// TIA Portal project "Rid TIA Pick & Place" (V15)
// Vorlageprojekt für das Buch mit Zielsystem S7-1200

(* hardware
DEVICE "S7-1200-Station_1"  S7-1200 Station
   slot 0: "Baugruppenträger_0"  Rack  V1.0
   slot 1: "PLC_1"  CPU 1211C DC/DC/DC  6ES7 211-1AE40-0XB0  V4.1
*)

// ===== PLC "PLC_1"  CPU 1211C DC/DC/DC =====

VAR_GLOBAL   // PLC tag table "Standard-Variablentabelle"
   "Clock_Byte" AT %MB0 : Byte;
   "Clock_10Hz" AT %M0.0 : Bool;
   "Clock_5Hz" AT %M0.1 : Bool;
   "Clock_2.5Hz" AT %M0.2 : Bool;
   "Clock_2Hz" AT %M0.3 : Bool;
   "Clock_1.25Hz" AT %M0.4 : Bool;
   "Clock_1Hz" AT %M0.5 : Bool;
   "Clock_0.625Hz" AT %M0.6 : Bool;
   "Clock_0.5Hz" AT %M0.7 : Bool;
END_VAR

VAR_GLOBAL   // PLC tag table "Assembler"
   "Item at entry" AT %I0.0 : Bool;
   "Item at exit" AT %I0.1 : Bool;
   "Moving X" AT %I0.2 : Bool;
   "Moving Z" AT %I0.3 : Bool;
   "Item detected" AT %I0.4 : Bool;
   "Start" AT %I0.5 : Bool;
   "Reset" AT %I0.6 : Bool;
   "Stop" AT %I0.7 : Bool;
   "Emergency stop" AT %I1.0 : Bool;
   "Auto" AT %I1.1 : Bool;
   "FACTORY I/O (Running)" AT %I1.2 : Bool;
   "Entry conveyor" AT %Q0.0 : Bool;
   "Exit conveyor" AT %Q0.1 : Bool;
   "Move X" AT %Q0.2 : Bool;
   "Move Z" AT %Q0.3 : Bool;
   "Grab" AT %Q0.4 : Bool;
   "Start light" AT %Q0.5 : Bool;
   "Reset light" AT %Q0.6 : Bool;
   "Stop light" AT %Q0.7 : Bool;
   "Counter" AT %QD30 : DInt;
END_VAR

VAR_GLOBAL   // PLC tag table "GRAFCET"
   "Reset Step" AT %M2.0 : Bool;   // memReset
   "All Step Off A" AT %M2.1 : Bool;   // memStepsOff
   "Initial Step A" AT %M2.2 : Bool;   // memInit
   "Step 1" AT %M2.3 : Bool;   // Step 1
   "Step 2" AT %M2.4 : Bool;   // Step 2
   "Step 3" AT %M2.5 : Bool;   // Step 3
   "Step 4" AT %M2.6 : Bool;   // Step 4
   "Step 5" AT %M2.7 : Bool;   // Step 5
   "Step 6" AT %M3.0 : Bool;   // Step 6
   "Step 7" AT %M3.1 : Bool;   // Step 7
   "Step 8" AT %M3.2 : Bool;   // Step 8
   "Step 9" AT %M3.3 : Bool;   // Step 9
   "Step 10" AT %M3.4 : Bool;   // Step 10
   "Auto Flag" AT %M6.0 : Bool;   // Auto Flag
   "N Moving Z 1" AT %M6.1 : Bool;
   "N Moving Z 2" AT %M6.2 : Bool;
   "N Moving z 3" AT %M6.3 : Bool;
   "N Moving X 1" AT %M6.4 : Bool;
   "N Item at entry" AT %M6.5 : Bool;
   "N Moving X 2" AT %M6.6 : Bool;
   "Step 11" AT %M3.5 : Bool;
   "N Moving z 4" AT %M6.7 : Bool;
   "N Moving X 3" AT %M7.0 : Bool;
   "Initial Step B" AT %M3.6 : Bool;
   "All Step Off B" AT %M3.7 : Bool;
   "Step 12" AT %M4.1 : Bool;
   "Step 13" AT %M4.2 : Bool;
   "Step 14" AT %M4.3 : Bool;
   "Step 15" AT %M4.4 : Bool;
   "N Moving z 5" AT %M7.2 : Bool;
   "N Moving z 6" AT %M7.3 : Bool;
END_VAR

// folder: System blocks/Program resources

DATA_BLOCK "Parts Counter"   // DB1
{ S7_Optimized_Access := 'TRUE' }
AUTHOR : Simatic
FAMILY : IEC
NAME : CNTR
VERSION : 1.0
// stored: InstanceOfName IEC_COUNTER
"IEC_COUNTER"
BEGIN
END_DATA_BLOCK

DATA_BLOCK "IEC_Timer_0_DB"   // DB2
{ S7_Optimized_Access := 'TRUE' }
AUTHOR : Simatic
FAMILY : IEC
NAME : IEC_TMR
VERSION : 1.0
// stored: InstanceOfName IEC_TIMER
"IEC_TIMER"
BEGIN
END_DATA_BLOCK

// folder: (top level)

FUNCTION "Steps" : Void   // FC1, LAD
{ S7_Optimized_Access := 'TRUE' }
VERSION : 0.1
   VAR_TEMP   // added for the SCL form of the ladder/FBD networks
      _w1 : Bool;
   END_VAR
BEGIN

REGION Network 1: Auto Flag
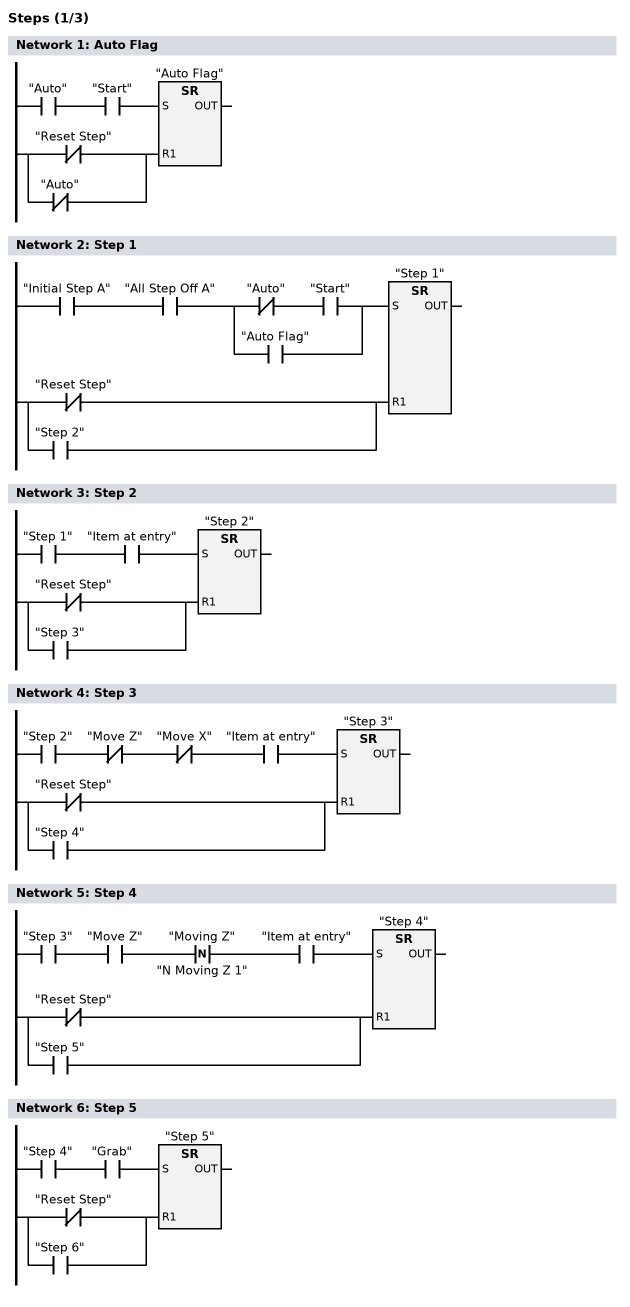
   RUNG wire#powerrail
      Contact( "Auto" )
      Contact( "Start" )
      S_SR(operand := "Auto Flag", r1 := wire#w1)
   END_RUNG
   RUNG wire#powerrail
      I_Contact( "Reset Step" )
   END_RUNG wire#w1
   RUNG wire#powerrail
      I_Contact( "Auto" )
   END_RUNG wire#w1
   // the same network as SCL:
   IF "Auto" AND "Start" THEN
       "Auto Flag" := TRUE;   // SR flip-flop
   END_IF;
   IF NOT "Reset Step" OR NOT "Auto" THEN "Auto Flag" := FALSE; END_IF;
END_REGION

REGION Network 2: Step 1
   RUNG wire#powerrail
      Contact( "Initial Step A" )
      Contact( "All Step Off A" )
      wire#w1
      I_Contact( "Auto" )
      Contact( "Start" )
      wire#w2
      S_SR(operand := "Step 1", r1 := wire#w3)
   END_RUNG
   RUNG wire#w1
      Contact( "Auto Flag" )
   END_RUNG wire#w2
   RUNG wire#powerrail
      I_Contact( "Reset Step" )
   END_RUNG wire#w3
   RUNG wire#powerrail
      Contact( "Step 2" )
   END_RUNG wire#w3
   // the same network as SCL:
   IF "Initial Step A" AND "All Step Off A" AND ((NOT "Auto" AND "Start") OR "Auto Flag") THEN
       "Step 1" := TRUE;   // SR flip-flop
   END_IF;
   IF NOT "Reset Step" OR "Step 2" THEN "Step 1" := FALSE; END_IF;
END_REGION

REGION Network 3: Step 2
   RUNG wire#powerrail
      Contact( "Step 1" )
      Contact( "Item at entry" )
      S_SR(operand := "Step 2", r1 := wire#w1)
   END_RUNG
   RUNG wire#powerrail
      I_Contact( "Reset Step" )
   END_RUNG wire#w1
   RUNG wire#powerrail
      Contact( "Step 3" )
   END_RUNG wire#w1
   // the same network as SCL:
   IF "Step 1" AND "Item at entry" THEN
       "Step 2" := TRUE;   // SR flip-flop
   END_IF;
   IF NOT "Reset Step" OR "Step 3" THEN "Step 2" := FALSE; END_IF;
END_REGION

REGION Network 4: Step 3
   RUNG wire#powerrail
      Contact( "Step 2" )
      I_Contact( "Move Z" )
      I_Contact( "Move X" )
      Contact( "Item at entry" )
      S_SR(operand := "Step 3", r1 := wire#w1)
   END_RUNG
   RUNG wire#powerrail
      I_Contact( "Reset Step" )
   END_RUNG wire#w1
   RUNG wire#powerrail
      Contact( "Step 4" )
   END_RUNG wire#w1
   // the same network as SCL:
   IF "Step 2" AND NOT "Move Z" AND NOT "Move X" AND "Item at entry" THEN
       "Step 3" := TRUE;   // SR flip-flop
   END_IF;
   IF NOT "Reset Step" OR "Step 4" THEN "Step 3" := FALSE; END_IF;
END_REGION

REGION Network 5: Step 4
   RUNG wire#powerrail
      Contact( "Step 3" )
      Contact( "Move Z" )
      N_Contact(operand := "Moving Z", bit := "N Moving Z 1")
      Contact( "Item at entry" )
      S_SR(operand := "Step 4", r1 := wire#w1)
   END_RUNG
   RUNG wire#powerrail
      I_Contact( "Reset Step" )
   END_RUNG wire#w1
   RUNG wire#powerrail
      Contact( "Step 5" )
   END_RUNG wire#w1
   // the same network as SCL:
   #_w1 := "Step 3" AND "Move Z" AND NOT "Moving Z" AND "N Moving Z 1";   // falling edge of "Moving Z"
   "N Moving Z 1" := "Moving Z";
   IF #_w1 AND "Item at entry" THEN
       "Step 4" := TRUE;   // SR flip-flop
   END_IF;
   IF NOT "Reset Step" OR "Step 5" THEN "Step 4" := FALSE; END_IF;
END_REGION

REGION Network 6: Step 5
   RUNG wire#powerrail
      Contact( "Step 4" )
      Contact( "Grab" )
      S_SR(operand := "Step 5", r1 := wire#w1)
   END_RUNG
   RUNG wire#powerrail
      I_Contact( "Reset Step" )
   END_RUNG wire#w1
   RUNG wire#powerrail
      Contact( "Step 6" )
   END_RUNG wire#w1
   // the same network as SCL:
   IF "Step 4" AND "Grab" THEN
       "Step 5" := TRUE;   // SR flip-flop
   END_IF;
   IF NOT "Reset Step" OR "Step 6" THEN "Step 5" := FALSE; END_IF;
END_REGION

REGION Network 7: Step 6
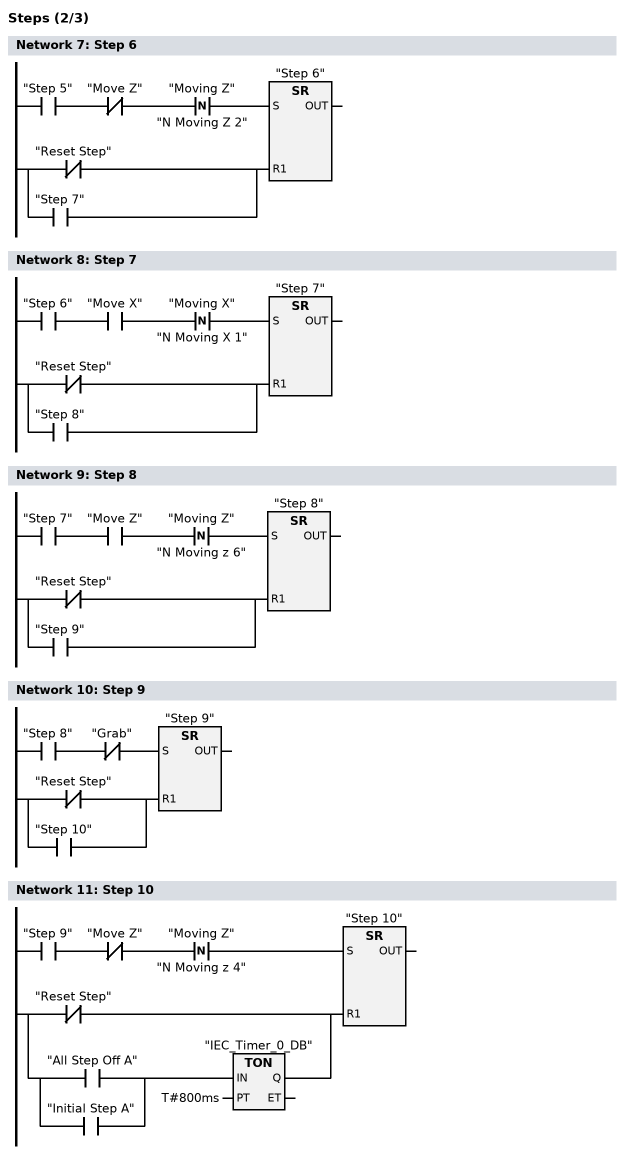
   RUNG wire#powerrail
      Contact( "Step 5" )
      I_Contact( "Move Z" )
      N_Contact(operand := "Moving Z", bit := "N Moving Z 2")
      S_SR(operand := "Step 6", r1 := wire#w1)
   END_RUNG
   RUNG wire#powerrail
      I_Contact( "Reset Step" )
   END_RUNG wire#w1
   RUNG wire#powerrail
      Contact( "Step 7" )
   END_RUNG wire#w1
   // the same network as SCL:
   #_w1 := "Step 5" AND NOT "Move Z" AND NOT "Moving Z" AND "N Moving Z 2";   // falling edge of "Moving Z"
   "N Moving Z 2" := "Moving Z";
   IF #_w1 THEN
       "Step 6" := TRUE;   // SR flip-flop
   END_IF;
   IF NOT "Reset Step" OR "Step 7" THEN "Step 6" := FALSE; END_IF;
END_REGION

REGION Network 8: Step 7
   RUNG wire#powerrail
      Contact( "Step 6" )
      Contact( "Move X" )
      N_Contact(operand := "Moving X", bit := "N Moving X 1")
      S_SR(operand := "Step 7", r1 := wire#w1)
   END_RUNG
   RUNG wire#powerrail
      I_Contact( "Reset Step" )
   END_RUNG wire#w1
   RUNG wire#powerrail
      Contact( "Step 8" )
   END_RUNG wire#w1
   // the same network as SCL:
   #_w1 := "Step 6" AND "Move X" AND NOT "Moving X" AND "N Moving X 1";   // falling edge of "Moving X"
   "N Moving X 1" := "Moving X";
   IF #_w1 THEN
       "Step 7" := TRUE;   // SR flip-flop
   END_IF;
   IF NOT "Reset Step" OR "Step 8" THEN "Step 7" := FALSE; END_IF;
END_REGION

REGION Network 9: Step 8
   RUNG wire#powerrail
      Contact( "Step 7" )
      Contact( "Move Z" )
      N_Contact(operand := "Moving Z", bit := "N Moving z 6")
      S_SR(operand := "Step 8", r1 := wire#w1)
   END_RUNG
   RUNG wire#powerrail
      I_Contact( "Reset Step" )
   END_RUNG wire#w1
   RUNG wire#powerrail
      Contact( "Step 9" )
   END_RUNG wire#w1
   // the same network as SCL:
   #_w1 := "Step 7" AND "Move Z" AND NOT "Moving Z" AND "N Moving z 6";   // falling edge of "Moving Z"
   "N Moving z 6" := "Moving Z";
   IF #_w1 THEN
       "Step 8" := TRUE;   // SR flip-flop
   END_IF;
   IF NOT "Reset Step" OR "Step 9" THEN "Step 8" := FALSE; END_IF;
END_REGION

REGION Network 10: Step 9
   RUNG wire#powerrail
      Contact( "Step 8" )
      I_Contact( "Grab" )
      S_SR(operand := "Step 9", r1 := wire#w1)
   END_RUNG
   RUNG wire#powerrail
      I_Contact( "Reset Step" )
   END_RUNG wire#w1
   RUNG wire#powerrail
      Contact( "Step 10" )
   END_RUNG wire#w1
   // the same network as SCL:
   IF "Step 8" AND NOT "Grab" THEN
       "Step 9" := TRUE;   // SR flip-flop
   END_IF;
   IF NOT "Reset Step" OR "Step 10" THEN "Step 9" := FALSE; END_IF;
END_REGION

REGION Network 11: Step 10
   #_w1 := "Step 9" AND NOT "Move Z" AND NOT "Moving Z" AND "N Moving z 4";   // falling edge of "Moving Z"
   "N Moving z 4" := "Moving Z";
   "IEC_Timer_0_DB".TON(IN := "All Step Off A" OR "Initial Step A", PT := T#800ms);
   IF #_w1 THEN
       "Step 10" := TRUE;   // SR flip-flop
   END_IF;
   IF NOT "Reset Step" OR "IEC_Timer_0_DB".Q THEN "Step 10" := FALSE; END_IF;
END_REGION

REGION Network 12: Step 11
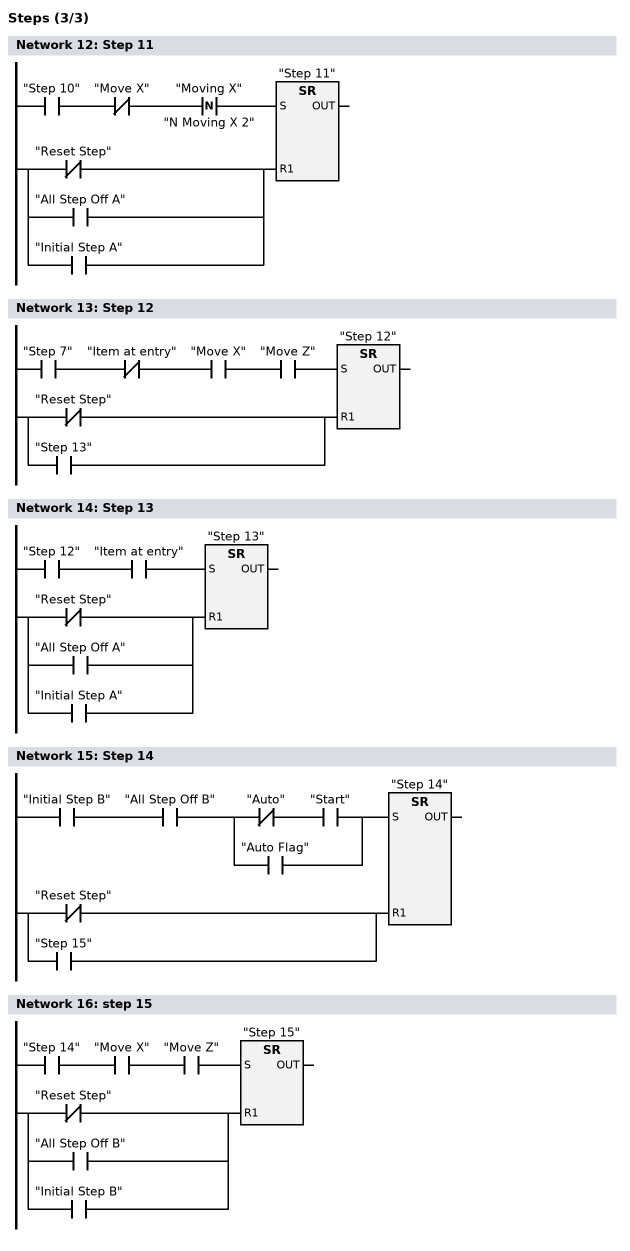
   RUNG wire#powerrail
      Contact( "Step 10" )
      I_Contact( "Move X" )
      N_Contact(operand := "Moving X", bit := "N Moving X 2")
      S_SR(operand := "Step 11", r1 := wire#w1)
   END_RUNG
   RUNG wire#powerrail
      I_Contact( "Reset Step" )
   END_RUNG wire#w1
   RUNG wire#powerrail
      Contact( "All Step Off A" )
   END_RUNG wire#w1
   RUNG wire#powerrail
      Contact( "Initial Step A" )
   END_RUNG wire#w1
   // the same network as SCL:
   #_w1 := "Step 10" AND NOT "Move X" AND NOT "Moving X" AND "N Moving X 2";   // falling edge of "Moving X"
   "N Moving X 2" := "Moving X";
   IF #_w1 THEN
       "Step 11" := TRUE;   // SR flip-flop
   END_IF;
   IF NOT "Reset Step" OR "All Step Off A" OR "Initial Step A" THEN "Step 11" := FALSE; END_IF;
END_REGION

REGION Network 13: Step 12
   RUNG wire#powerrail
      Contact( "Step 7" )
      I_Contact( "Item at entry" )
      Contact( "Move X" )
      Contact( "Move Z" )
      S_SR(operand := "Step 12", r1 := wire#w1)
   END_RUNG
   RUNG wire#powerrail
      I_Contact( "Reset Step" )
   END_RUNG wire#w1
   RUNG wire#powerrail
      Contact( "Step 13" )
   END_RUNG wire#w1
   // the same network as SCL:
   IF "Step 7" AND NOT "Item at entry" AND "Move X" AND "Move Z" THEN
       "Step 12" := TRUE;   // SR flip-flop
   END_IF;
   IF NOT "Reset Step" OR "Step 13" THEN "Step 12" := FALSE; END_IF;
END_REGION

REGION Network 14: Step 13
   RUNG wire#powerrail
      Contact( "Step 12" )
      Contact( "Item at entry" )
      S_SR(operand := "Step 13", r1 := wire#w1)
   END_RUNG
   RUNG wire#powerrail
      I_Contact( "Reset Step" )
   END_RUNG wire#w1
   RUNG wire#powerrail
      Contact( "All Step Off A" )
   END_RUNG wire#w1
   RUNG wire#powerrail
      Contact( "Initial Step A" )
   END_RUNG wire#w1
   // the same network as SCL:
   IF "Step 12" AND "Item at entry" THEN
       "Step 13" := TRUE;   // SR flip-flop
   END_IF;
   IF NOT "Reset Step" OR "All Step Off A" OR "Initial Step A" THEN "Step 13" := FALSE; END_IF;
END_REGION

REGION Network 15: Step 14
   RUNG wire#powerrail
      Contact( "Initial Step B" )
      Contact( "All Step Off B" )
      wire#w1
      I_Contact( "Auto" )
      Contact( "Start" )
      wire#w2
      S_SR(operand := "Step 14", r1 := wire#w3)
   END_RUNG
   RUNG wire#w1
      Contact( "Auto Flag" )
   END_RUNG wire#w2
   RUNG wire#powerrail
      I_Contact( "Reset Step" )
   END_RUNG wire#w3
   RUNG wire#powerrail
      Contact( "Step 15" )
   END_RUNG wire#w3
   // the same network as SCL:
   IF "Initial Step B" AND "All Step Off B" AND ((NOT "Auto" AND "Start") OR "Auto Flag") THEN
       "Step 14" := TRUE;   // SR flip-flop
   END_IF;
   IF NOT "Reset Step" OR "Step 15" THEN "Step 14" := FALSE; END_IF;
END_REGION

REGION Network 16: step 15
   RUNG wire#powerrail
      Contact( "Step 14" )
      Contact( "Move X" )
      Contact( "Move Z" )
      S_SR(operand := "Step 15", r1 := wire#w1)
   END_RUNG
   RUNG wire#powerrail
      I_Contact( "Reset Step" )
   END_RUNG wire#w1
   RUNG wire#powerrail
      Contact( "All Step Off B" )
   END_RUNG wire#w1
   RUNG wire#powerrail
      Contact( "Initial Step B" )
   END_RUNG wire#w1
   // the same network as SCL:
   IF "Step 14" AND "Move X" AND "Move Z" THEN
       "Step 15" := TRUE;   // SR flip-flop
   END_IF;
   IF NOT "Reset Step" OR "All Step Off B" OR "Initial Step B" THEN "Step 15" := FALSE; END_IF;
END_REGION
END_FUNCTION

FUNCTION "Actions" : Void   // FC2, LAD
{ S7_Optimized_Access := 'TRUE' }
VERSION : 0.1
BEGIN

REGION Network 1: Entry conveyor
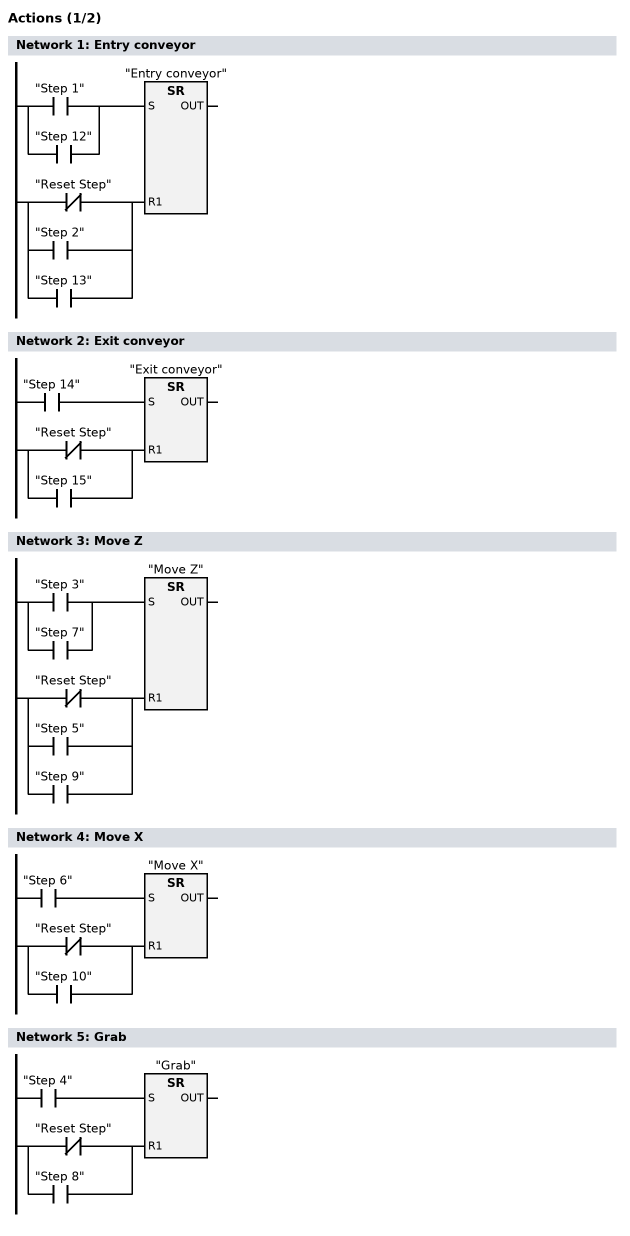
   RUNG wire#powerrail
      Contact( "Step 1" )
      wire#w1
      S_SR(operand := "Entry conveyor", r1 := wire#w2)
   END_RUNG
   RUNG wire#powerrail
      Contact( "Step 12" )
   END_RUNG wire#w1
   RUNG wire#powerrail
      I_Contact( "Reset Step" )
   END_RUNG wire#w2
   RUNG wire#powerrail
      Contact( "Step 2" )
   END_RUNG wire#w2
   RUNG wire#powerrail
      Contact( "Step 13" )
   END_RUNG wire#w2
   // the same network as SCL:
   IF "Step 1" OR "Step 12" THEN
       "Entry conveyor" := TRUE;   // SR flip-flop
   END_IF;
   IF NOT "Reset Step" OR "Step 2" OR "Step 13" THEN "Entry conveyor" := FALSE; END_IF;
END_REGION

REGION Network 2: Exit conveyor
   RUNG wire#powerrail
      Contact( "Step 14" )
      S_SR(operand := "Exit conveyor", r1 := wire#w1)
   END_RUNG
   RUNG wire#powerrail
      I_Contact( "Reset Step" )
   END_RUNG wire#w1
   RUNG wire#powerrail
      Contact( "Step 15" )
   END_RUNG wire#w1
   // the same network as SCL:
   IF "Step 14" THEN
       "Exit conveyor" := TRUE;   // SR flip-flop
   END_IF;
   IF NOT "Reset Step" OR "Step 15" THEN "Exit conveyor" := FALSE; END_IF;
END_REGION

REGION Network 3: Move Z
   RUNG wire#powerrail
      Contact( "Step 3" )
      wire#w1
      S_SR(operand := "Move Z", r1 := wire#w2)
   END_RUNG
   RUNG wire#powerrail
      Contact( "Step 7" )
   END_RUNG wire#w1
   RUNG wire#powerrail
      I_Contact( "Reset Step" )
   END_RUNG wire#w2
   RUNG wire#powerrail
      Contact( "Step 5" )
   END_RUNG wire#w2
   RUNG wire#powerrail
      Contact( "Step 9" )
   END_RUNG wire#w2
   // the same network as SCL:
   IF "Step 3" OR "Step 7" THEN
       "Move Z" := TRUE;   // SR flip-flop
   END_IF;
   IF NOT "Reset Step" OR "Step 5" OR "Step 9" THEN "Move Z" := FALSE; END_IF;
END_REGION

REGION Network 4: Move X
   RUNG wire#powerrail
      Contact( "Step 6" )
      S_SR(operand := "Move X", r1 := wire#w1)
   END_RUNG
   RUNG wire#powerrail
      I_Contact( "Reset Step" )
   END_RUNG wire#w1
   RUNG wire#powerrail
      Contact( "Step 10" )
   END_RUNG wire#w1
   // the same network as SCL:
   IF "Step 6" THEN
       "Move X" := TRUE;   // SR flip-flop
   END_IF;
   IF NOT "Reset Step" OR "Step 10" THEN "Move X" := FALSE; END_IF;
END_REGION

REGION Network 5: Grab
   RUNG wire#powerrail
      Contact( "Step 4" )
      S_SR(operand := "Grab", r1 := wire#w1)
   END_RUNG
   RUNG wire#powerrail
      I_Contact( "Reset Step" )
   END_RUNG wire#w1
   RUNG wire#powerrail
      Contact( "Step 8" )
   END_RUNG wire#w1
   // the same network as SCL:
   IF "Step 4" THEN
       "Grab" := TRUE;   // SR flip-flop
   END_IF;
   IF NOT "Reset Step" OR "Step 8" THEN "Grab" := FALSE; END_IF;
END_REGION

REGION Network 6: Parts Counter
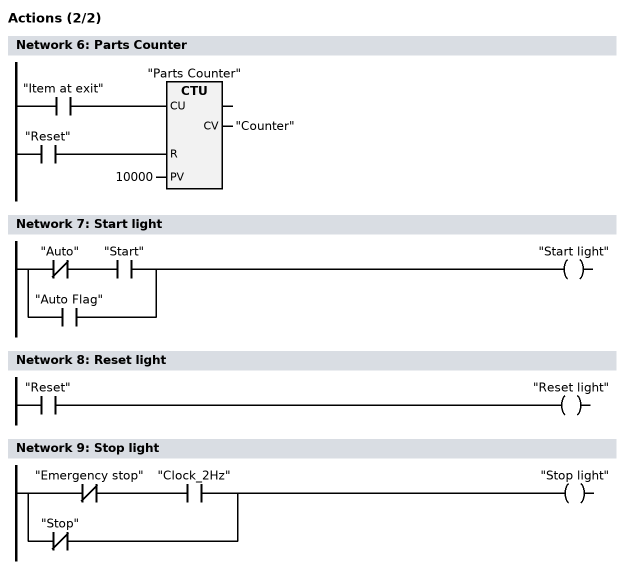
   "Parts Counter".CTU(CU := "Item at exit", R := "Reset", PV := 10000, CV => "Counter");
END_REGION

REGION Network 7: Start light
   RUNG wire#powerrail
      I_Contact( "Auto" )
      Contact( "Start" )
      wire#w1
      Coil( "Start light" )
   END_RUNG
   RUNG wire#powerrail
      Contact( "Auto Flag" )
   END_RUNG wire#w1
   // the same network as SCL:
   "Start light" := (NOT "Auto" AND "Start") OR "Auto Flag";
END_REGION

REGION Network 8: Reset light
   RUNG wire#powerrail
      Contact( "Reset" )
      Coil( "Reset light" )
   END_RUNG
   // the same network as SCL:
   "Reset light" := "Reset";
END_REGION

REGION Network 9: Stop light
   RUNG wire#powerrail
      I_Contact( "Emergency stop" )
      Contact( "Clock_2Hz" )
      wire#w1
      Coil( "Stop light" )
   END_RUNG
   RUNG wire#powerrail
      I_Contact( "Stop" )
   END_RUNG wire#w1
   // the same network as SCL:
   "Stop light" := (NOT "Emergency stop" AND "Clock_2Hz") OR NOT "Stop";
END_REGION
END_FUNCTION

FUNCTION "MHJ-PLC-Lab-Function-S71200" : Void   // FC9000, SCL
{ S7_Optimized_Access := 'TRUE' }
VERSION : 0.1
   VAR_TEMP
      rdTimeReturn : Int;
      outputTime : DTL;
      SyncVal : Byte;
      forVal : Int;
      forVal_2 : Int;
      Value : Byte;
   END_VAR
   VAR CONSTANT
      CompVal : Byte := 16#34;
      Value_01 : Byte := 16#11;
      Value_01_DW : DWord := 16#A165_D992;
      Value_02_DW : DWord := 16#58BE_4401;
   END_VAR
BEGIN

   #Value:=PEEK(area := 16#82,
        dbNumber := 0,
        byteOffset := 511);
   #Value := #Value + 1;

   POKE(area := 16#82,
        dbNumber := 0,
        byteOffset := 511,
        value := #Value);

   POKE(area:=16#81,
        dbNumber:=0,
        byteOffset:=1016,
        value:=#Value_01_DW);
   POKE(area := 16#81,
        dbNumber := 0,
        byteOffset := 1020,
        value := #Value_02_DW);

   POKE(area := 16#81,
        dbNumber := 0,
        byteOffset := 511,
        value := B#16#00);

   FOR #forVal := 0 TO 120 DO
       FOR #forVal_2:=0 TO 10 DO
           #rdTimeReturn:=RD_SYS_T(#outputTime);
           #rdTimeReturn := WR_SYS_T(#outputTime);
           #rdTimeReturn := RD_SYS_T(#outputTime);
           #rdTimeReturn := WR_SYS_T(#outputTime);
       END_FOR;
       #SyncVal:= PEEK(area := 16#81,
                      dbNumber := 0,
                      byteOffset := 511);
       IF #SyncVal = #CompVal THEN
          GOTO M_1;
       END_IF;
   END_FOR;
   RETURN;

   M_1:
   POKE(area := 16#81,
        dbNumber := 0,
        byteOffset := 511,
        value := B#16#0);
END_FUNCTION

ORGANIZATION_BLOCK "Main"   // OB1, LAD, ProgramCycle
TITLE = "Main Program Sweep (Cycle)"
{ S7_Optimized_Access := 'TRUE' }
VERSION : 0.1
   VAR_INPUT
      Initial_Call : Bool;   // Initial call of this OB
      Remanence : Bool;   // =True, if remanent data are available
   END_VAR
BEGIN

REGION Network 1: Konnektierungsbaustein für PLC-Lab / Factory IO Template
   // Im Netzwerk 1 wird der Konnektierungsbaustein für PLC-Lab aufgerufen.
   // Dieser Aufruf darf nicht entfernt werden!
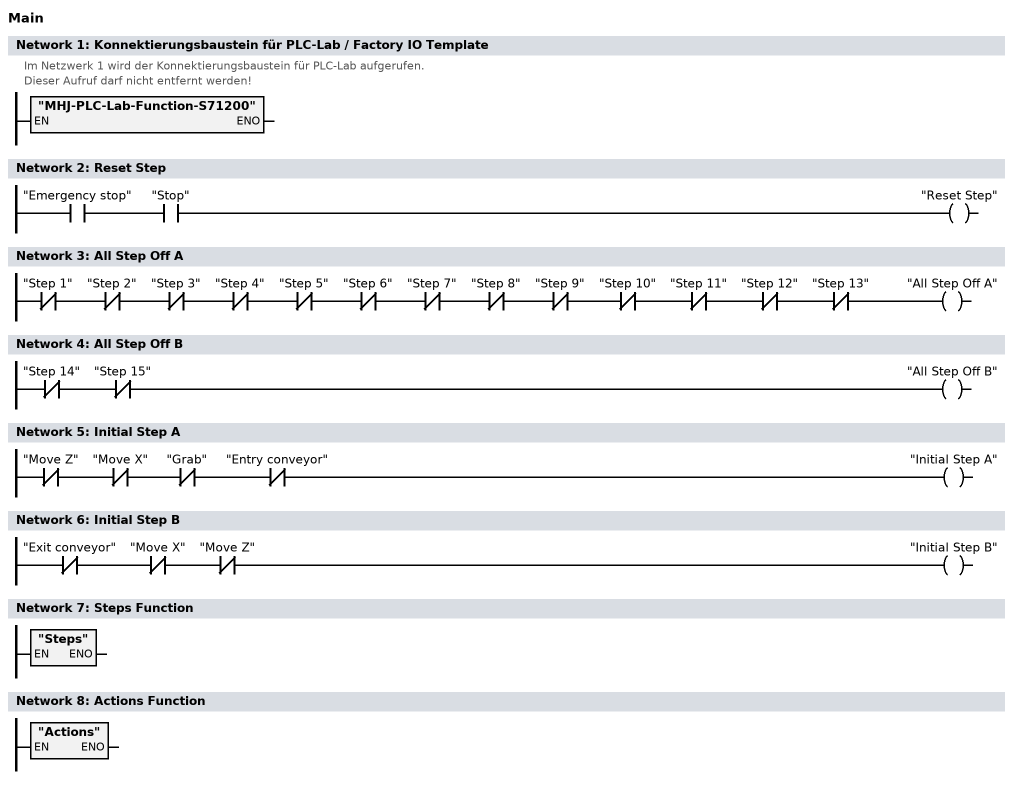
   RUNG wire#powerrail
      "MHJ-PLC-Lab-Function-S71200"()
   END_RUNG
   // the same network as SCL:
   "MHJ-PLC-Lab-Function-S71200"();
END_REGION

REGION Network 2: Reset Step
   RUNG wire#powerrail
      Contact( "Emergency stop" )
      Contact( "Stop" )
      Coil( "Reset Step" )
   END_RUNG
   // the same network as SCL:
   "Reset Step" := "Emergency stop" AND "Stop";
END_REGION

REGION Network 3: All Step Off A
   RUNG wire#powerrail
      I_Contact( "Step 1" )
      I_Contact( "Step 2" )
      I_Contact( "Step 3" )
      I_Contact( "Step 4" )
      I_Contact( "Step 5" )
      I_Contact( "Step 6" )
      I_Contact( "Step 7" )
      I_Contact( "Step 8" )
      I_Contact( "Step 9" )
      I_Contact( "Step 10" )
      I_Contact( "Step 11" )
      I_Contact( "Step 12" )
      I_Contact( "Step 13" )
      Coil( "All Step Off A" )
   END_RUNG
   // the same network as SCL:
   "All Step Off A" := NOT "Step 1" AND NOT "Step 2" AND NOT "Step 3" AND NOT "Step 4" AND NOT "Step 5" AND NOT "Step 6" AND NOT "Step 7" AND NOT "Step 8" AND NOT "Step 9" AND NOT "Step 10" AND NOT "Step 11" AND NOT "Step 12" AND NOT "Step 13";
END_REGION

REGION Network 4: All Step Off B
   RUNG wire#powerrail
      I_Contact( "Step 14" )
      I_Contact( "Step 15" )
      Coil( "All Step Off B" )
   END_RUNG
   // the same network as SCL:
   "All Step Off B" := NOT "Step 14" AND NOT "Step 15";
END_REGION

REGION Network 5: Initial Step A
   RUNG wire#powerrail
      I_Contact( "Move Z" )
      I_Contact( "Move X" )
      I_Contact( "Grab" )
      I_Contact( "Entry conveyor" )
      Coil( "Initial Step A" )
   END_RUNG
   // the same network as SCL:
   "Initial Step A" := NOT "Move Z" AND NOT "Move X" AND NOT "Grab" AND NOT "Entry conveyor";
END_REGION

REGION Network 6: Initial Step B
   RUNG wire#powerrail
      I_Contact( "Exit conveyor" )
      I_Contact( "Move X" )
      I_Contact( "Move Z" )
      Coil( "Initial Step B" )
   END_RUNG
   // the same network as SCL:
   "Initial Step B" := NOT "Exit conveyor" AND NOT "Move X" AND NOT "Move Z";
END_REGION

REGION Network 7: Steps Function
   RUNG wire#powerrail
      "Steps"()
   END_RUNG
   // the same network as SCL:
   "Steps"();
END_REGION

REGION Network 8: Actions Function
   RUNG wire#powerrail
      "Actions"()
   END_RUNG
   // the same network as SCL:
   "Actions"();
END_REGION
END_ORGANIZATION_BLOCK